Fanuc KAREL source: kx00001.KL

-- PROVISIONAL review KL for V770-1; original PC SHA256 c5563e454bf2d4dba3e591bf9e6ad35b98e6644c9411b64773526873295e4de7
-- Incomplete behavior may be omitted. Consult companion uncertainty JSON. Do not deploy.
PROGRAM KX00001
%NOLOCKGROUP
VAR
  I : INTEGER
  J : INTEGER
  B : BOOLEAN
  F : FILE
  S : STRING[80]
-- UNRESOLVED_DECL P type=000102
BEGIN
  -- UNRESOLVED_PC offsets 5-32; opcodes 22,3F,3F,3D
  -- UNRESOLVED_PC offsets 37-41; opcodes 7F
END KX00001
